FUNCTION_BLOCK AUDI_RampLimitFS (* Wrapper around RampLimitFS with AUDI load socket, AUDI out plug, and two AX status plugs (qAtZero, qAtFull) latched via E_D_FF *)
  (* Standard: 61499-2; Description: Copyright (c) 2026 Meisterschulen am Ostbahnhof This program and the accompanying materials are made available under the terms of the Eclipse Public License 2.0 which is available at https://www.eclipse.org/legal/epl-2.0/ SPDX-License-Identifier: EPL-2.0 *)
  (* Version 1.0, 2026-09-10, Franz Höpfinger, Meisterschulen am Ostbahnhof, initial API and implementation and/or initial documentation *)
  PACKAGE adapter::signalprocessing::ramp;
  IMPORT eclipse4diac::signalprocessing::RampLimitFS;
  IMPORT iec61131::conversion::F_UDINT_TO_DINT;
  IMPORT iec61131::conversion::F_DINT_TO_UDINT;
  IMPORT iec61499::events::E_D_FF;
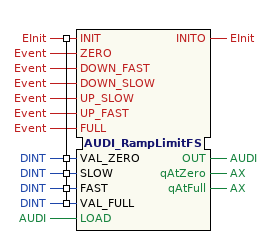
  EVENT_INPUT
    INIT : EInit WITH VAL_ZERO, SLOW, FAST, VAL_FULL; (* Initialization Request *)
    ZERO; (* Jump to VAL_ZERO *)
    DOWN_FAST; (* Ramp down fast *)
    DOWN_SLOW; (* Ramp down slow *)
    UP_SLOW; (* Ramp up slow *)
    UP_FAST; (* Ramp up fast *)
    FULL; (* Jump to VAL_FULL *)
  END_EVENT
  EVENT_OUTPUT
    INITO : EInit; (* Initialization Confirm *)
  END_EVENT
  VAR_INPUT
    VAL_ZERO : DINT := 0; (* Minimum value (default 0) *)
    SLOW : DINT := 1; (* Slow step size per cycle (default 1) *)
    FAST : DINT := 10; (* Fast step size per cycle (default 10) *)
    VAL_FULL : DINT := 100; (* Maximum value (default 100) *)
  END_VAR
  SOCKETS
    LOAD : adapter::types::unidirectional::AUDI; (* LOAD event and PV value as AUDI adapter socket *)
  END_SOCKETS
  PLUGS
    OUT : adapter::types::unidirectional::AUDI; (* Ramped output value as AUDI adapter plug *)
    qAtZero : adapter::types::unidirectional::AX; (* TRUE when OUT is at VAL_ZERO, latched via E_D_FF *)
    qAtFull : adapter::types::unidirectional::AX; (* TRUE when OUT is at VAL_FULL, latched via E_D_FF *)
  END_PLUGS
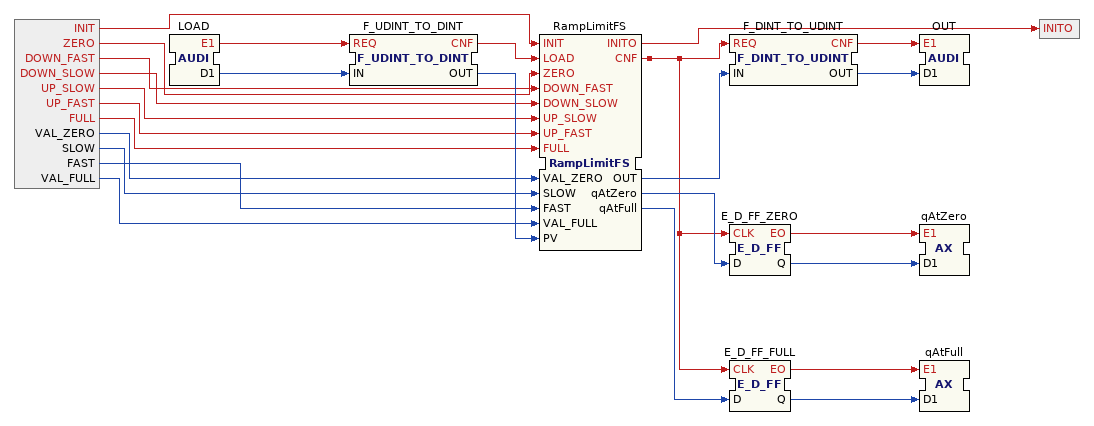
  FBS
    RampLimitFS : eclipse4diac::signalprocessing::RampLimitFS;
    F_UDINT_TO_DINT : iec61131::conversion::F_UDINT_TO_DINT;
    F_DINT_TO_UDINT : iec61131::conversion::F_DINT_TO_UDINT;
    E_D_FF_ZERO : iec61499::events::E_D_FF;
    E_D_FF_FULL : iec61499::events::E_D_FF;
  END_FBS
  EVENT_CONNECTIONS
    INIT TO RampLimitFS.INIT;
    RampLimitFS.INITO TO INITO;
    LOAD.E1 TO F_UDINT_TO_DINT.REQ;
    F_UDINT_TO_DINT.CNF TO RampLimitFS.LOAD;
    ZERO TO RampLimitFS.ZERO;
    DOWN_FAST TO RampLimitFS.DOWN_FAST;
    DOWN_SLOW TO RampLimitFS.DOWN_SLOW;
    UP_SLOW TO RampLimitFS.UP_SLOW;
    UP_FAST TO RampLimitFS.UP_FAST;
    FULL TO RampLimitFS.FULL;
    RampLimitFS.CNF TO F_DINT_TO_UDINT.REQ;
    F_DINT_TO_UDINT.CNF TO OUT.E1;
    RampLimitFS.CNF TO E_D_FF_ZERO.CLK;
    E_D_FF_ZERO.EO TO qAtZero.E1;
    RampLimitFS.CNF TO E_D_FF_FULL.CLK;
    E_D_FF_FULL.EO TO qAtFull.E1;
  END_CONNECTIONS
  DATA_CONNECTIONS
    VAL_ZERO TO RampLimitFS.VAL_ZERO;
    SLOW TO RampLimitFS.SLOW;
    FAST TO RampLimitFS.FAST;
    VAL_FULL TO RampLimitFS.VAL_FULL;
    LOAD.D1 TO F_UDINT_TO_DINT.IN;
    F_UDINT_TO_DINT.OUT TO RampLimitFS.PV;
    RampLimitFS.OUT TO F_DINT_TO_UDINT.IN;
    F_DINT_TO_UDINT.OUT TO OUT.D1;
    RampLimitFS.qAtZero TO E_D_FF_ZERO.D;
    E_D_FF_ZERO.Q TO qAtZero.D1;
    RampLimitFS.qAtFull TO E_D_FF_FULL.D;
    E_D_FF_FULL.Q TO qAtFull.D1;
  END_CONNECTIONS
END_FUNCTION_BLOCK
